FUNCTION Call_Aufzug

instFBElevator(
	CurrentPosition:= AufzugIstwert, 
	SensorOutfeed:= AufzugSensorAuslaufFoerderband, 
	SensorInfeed:= AufzugSensorEinlaufFoerderband, 
	ActorInstanceIndex := 0,
	ActorInstanceName := 'Zufuehrung',
	HMIInterface := HMI.hmiMachineSectionInterface,
	SetPointPositionElevator=> AufzugSollwert, 
	ConveyorForward=> AufzugFoerderbandVorwaerts, 
	ConveyorBackward=> AufzugFoerderbandRueckwaerts, 
	ElevatorInPosition=> AufzugInPosition, 
	OperatingMode:= instOperatingMode.StateOperatingMode);
	
instFBElevator.MoveElevator(AufzugBewegen, SollPosition);
instFBElevator.ConveyorForward_ON(AufzugFoerderbandVor);
instFBElevator.ConveyorBackward_ON(AufzugFoerderbandRueck);
instFBElevator.Conveyor_OFF(AufzugFoerderbandStop);

END_FUNCTION

(* stored: Version 1.1.0.1
   POU Call_Aufzug: Id {aacc9d31-4429-4f84-b695-0be7a89ff098}, SpecialFunc None *)
